FUNCTION_BLOCK FB_ManualControl
VAR_INPUT
	eMode : E_Mode;
	eStatus : E_Status;
	stParam : ST_Parameters;
END_VAR
VAR_OUTPUT
	fControlOutputNormalizedCylinder : LREAL;
	fControlOutputNormalizedWinch : LREAL;
END_VAR
	
VAR
	fbJoystick : FB_Joystick;
	fbOpenLoopCylindeControl : FB_OpenLoopCylinderControl;
	fbOpenLoopWinchControl : FB_OpenLoopWinchControl;
END_VAR

IF NOT(G_RawSensorData.bJoystickEnable) THEN
	fbJoystick(
		bEnable := (eMode = E_Mode.Manual),
		stParam := stParam,
		fNormalizedInput := G_ScaledSensorData.fJoystickNormalizedX,
	);
	
	fbOpenLoopCylindeControl(
		bEnable := (eMode = E_Mode.Manual),
		stParam := stParam,
		fInput_ms := fbJoystick.fOutput,
		fNormalizedOutput => fControlOutputNormalizedCylinder,
	);
	
	fbOpenLoopWinchControl(
		bEnable := (eMode = E_Mode.Manual),
		stParam := stParam,
		fInput_ms := 0.0,
		fNormalizedOutput => fControlOutputNormalizedWinch,
	);
	
ELSIF	(G_RawSensorData.bJoystickEnable) THEN
	fbJoystick(
		bEnable := (eMode = E_Mode.Manual),
		stParam := stParam,
		fNormalizedInput := G_ScaledSensorData.fJoystickNormalizedY
	);
	
	fbOpenLoopCylindeControl(
		bEnable := (eMode = E_Mode.Manual),
		stParam := stParam,
		fInput_ms := 0.0,
		fNormalizedOutput => fControlOutputNormalizedCylinder,
	);
	
	fbOpenLoopWinchControl(
		bEnable := (eMode = E_Mode.Manual),
		stParam := stParam,
		fInput_ms := fbJoystick.fOutput,
		fNormalizedOutput => fControlOutputNormalizedWinch,
	);
END_IF

END_FUNCTION_BLOCK

(* stored: Version 1.1.0.1, ProductVersion 3.1.4024.12
   POU FB_ManualControl: Id {030c0b1e-cfb9-4458-97b6-7b35e272d107}, SpecialFunc None *)
